// TIA Portal project "Estampado automatizado" (V17)
// Vorlageprojekt für das Buch mit Zielsystem S7-1200

(* hardware
DEVICE "S7-1200-Station_1"  S7-1200 Station
   slot 0: "Baugruppenträger_0"  Rack  V1.0
   slot 1: "PLC_1"  CPU 1211C DC/DC/DC  6ES7 211-1AE40-0XB0  V4.1
*)

// ===== PLC "PLC_1"  CPU 1211C DC/DC/DC =====

VAR_GLOBAL   // PLC tag table "02_Sensores"
   "Sensor_deteccion" AT %I0.3 : Bool;   // Sensor que detecta las bolsas
   "FC X+" AT %I0.4 : Bool;   // Final de carrera del cilindro de impresión extendido
   "FC X-" AT %I0.5 : Bool;   // Final de carrera del cilindro de impresión retraído
   "FC Z+" AT %I0.6 : Bool;   // Final de carrera del cilindro de sellado extendido
   "FC Z-" AT %I0.7 : Bool;   // Final de carrera del cilindro de sellado retraído
   "Sensor_conteo_final" AT %I1.0 : Bool;   // Sensor que detecta las bolsas al final del tunel
END_VAR

VAR_GLOBAL   // PLC tag table "01_Botones y selectores"
   "START" AT %I0.0 : Bool;   // Boton de START
   "STOP" AT %I0.1 : Bool;   // Boton de STOP
   "STOP_EMERGENCIA" AT %I0.2 : Bool;   // Boton enclavado de Parada de Emergencia
   "RESET_CONTEO" AT %I1.1 : Bool;   // Pulsador que reinicia el conteo
END_VAR

VAR_GLOBAL   // PLC tag table "03_Actuadores"
   "Motor_faja" AT %Q0.0 : Bool;   // Motor de la Faja Transportadora
   "EV mov Z" AT %Q0.2 : Bool;   // Electrovalvula Cilindro Eje Z Simple Efecto
   "EV mov X" AT %Q0.1 : Bool;   // Electrovalvula Cilindro Eje X Simple Efecto
   "Motor_faja_2" AT %Q0.6 : Bool;   // Motor de la Faja Transportadora (solo para simulacion)
END_VAR

VAR_GLOBAL   // PLC tag table "04_Luces e indicadores"
   "piloto_start" AT %Q0.3 : Bool;   // Luz indicadora de Proceso en Marcha
   "piloto_stop" AT %Q0.4 : Bool;   // Luz indicadora de Proceso Detenido
   "luz_emergencia" AT %Q0.5 : Bool;   // Luz indicadora de Parada de Emergencia
   "conteo_bolsas" AT %QW30 : Word;   // Cuenta las bolsas que terminan de pasar por el tunel de secado
END_VAR

VAR_GLOBAL   // PLC tag table "00_Variables_de_memoria"
   "Marcha" AT %M0.0 : Bool;   // Variable de memoria Proceso en Marcha
   "E0" AT %M0.1 : Bool;   // Variable de memoria Etapa 0 - inicio
   "E1" AT %M0.2 : Bool;   // Variable de memoria Etapa 1
   "E2" AT %M0.3 : Bool;   // Variable de memoria Etapa 2
   "E3" AT %M0.4 : Bool;   // Variable de memoria Etapa 3
   "E4" AT %M0.5 : Bool;   // Variable de memoria Etapa 4
   "E5" AT %M0.6 : Bool;   // Variable de memoria Etapa 5
   "E6" AT %M0.7 : Bool;   // Variable de memoria Etapa 6
END_VAR

// folder: System blocks/Program resources

DATA_BLOCK "IEC_Counter_0_DB"   // DB1
{ S7_Optimized_Access := 'TRUE' }
AUTHOR : Simatic
FAMILY : IEC
NAME : CNTR
VERSION : 1.0
// stored: InstanceOfName IEC_COUNTER
"IEC_COUNTER"
BEGIN
END_DATA_BLOCK

// folder: (top level)

FUNCTION "MHJ-PLC-Lab-Function-S71200" : Void   // FC9000, SCL
{ S7_Optimized_Access := 'TRUE' }
VERSION : 0.1
   VAR_TEMP
      rdTimeReturn : Int;
      outputTime : DTL;
      SyncVal : Byte;
      forVal : Int;
      forVal_2 : Int;
      Value : Byte;
   END_VAR
   VAR CONSTANT
      CompVal : Byte := 16#34;
      Value_01 : Byte := 16#11;
      Value_01_DW : DWord := 16#A165_D992;
      Value_02_DW : DWord := 16#58BE_4401;
   END_VAR
BEGIN

   #Value:=PEEK(area := 16#82,
        dbNumber := 0,
        byteOffset := 511);
   #Value := #Value + 1;

   POKE(area := 16#82,
        dbNumber := 0,
        byteOffset := 511,
        value := #Value);

   POKE(area:=16#81,
        dbNumber:=0,
        byteOffset:=1016,
        value:=#Value_01_DW);
   POKE(area := 16#81,
        dbNumber := 0,
        byteOffset := 1020,
        value := #Value_02_DW);

   POKE(area := 16#81,
        dbNumber := 0,
        byteOffset := 511,
        value := B#16#00);

   FOR #forVal := 0 TO 120 DO
       FOR #forVal_2:=0 TO 10 DO
           #rdTimeReturn:=RD_SYS_T(#outputTime);
           #rdTimeReturn := WR_SYS_T(#outputTime);
           #rdTimeReturn := RD_SYS_T(#outputTime);
           #rdTimeReturn := WR_SYS_T(#outputTime);
       END_FOR;
       #SyncVal:= PEEK(area := 16#81,
                      dbNumber := 0,
                      byteOffset := 511);
       IF #SyncVal = #CompVal THEN
          GOTO M_1;
       END_IF;
   END_FOR;
   RETURN;

   M_1:
   POKE(area := 16#81,
        dbNumber := 0,
        byteOffset := 511,
        value := B#16#0);
END_FUNCTION

ORGANIZATION_BLOCK "Main"   // OB1, LAD, ProgramCycle
TITLE = "Main Program Sweep (Cycle)"
{ S7_Optimized_Access := 'TRUE' }
VERSION : 0.1
   VAR_INPUT
      Initial_Call : Bool;   // Initial call of this OB
      Remanence : Bool;   // =True, if remanent data are available
   END_VAR
BEGIN

REGION Network 1: Konnektierungsbaustein für PLC-Lab / Bloque de conexion con Factory IO
   // Im Netzwerk 1 wird der Konnektierungsbaustein für PLC-Lab aufgerufen.
   // Dieser Aufruf darf nicht entfernt werden!
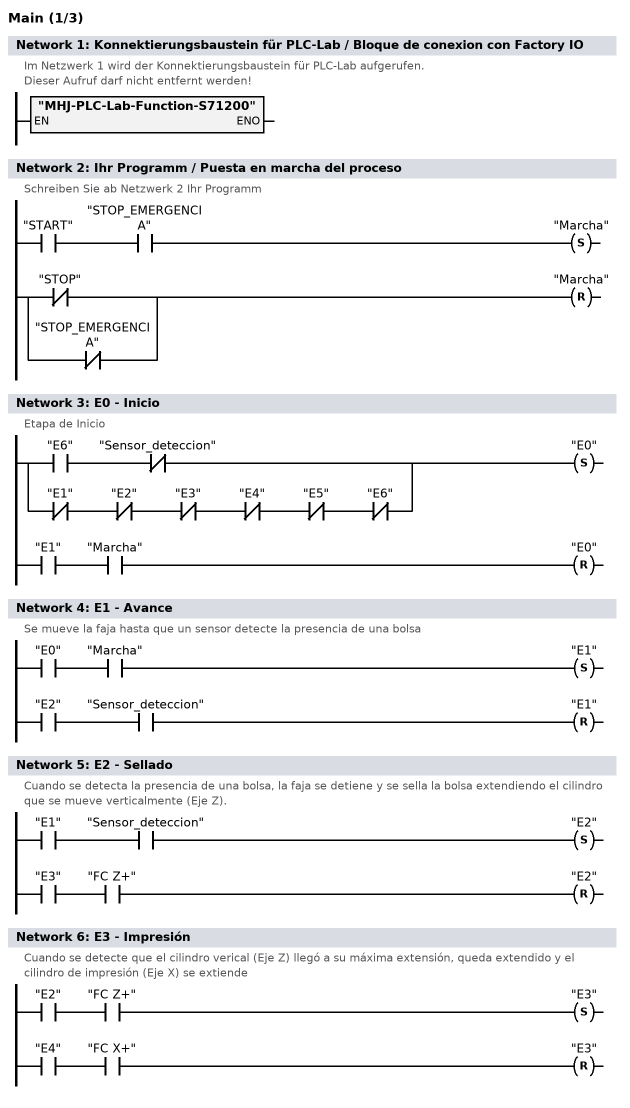
   RUNG wire#powerrail
      "MHJ-PLC-Lab-Function-S71200"()
   END_RUNG
   // the same network as SCL:
   "MHJ-PLC-Lab-Function-S71200"();
END_REGION

REGION Network 2: Ihr Programm / Puesta en marcha del proceso
   // Schreiben Sie ab Netzwerk 2 Ihr Programm
   RUNG wire#powerrail
      Contact( "START" )
      Contact( "STOP_EMERGENCIA" )
      S_Coil( "Marcha" )
   END_RUNG
   RUNG wire#powerrail
      I_Contact( "STOP" )
      wire#w1
      R_Coil( "Marcha" )
   END_RUNG
   RUNG wire#powerrail
      I_Contact( "STOP_EMERGENCIA" )
   END_RUNG wire#w1
   // the same network as SCL:
   IF "START" AND "STOP_EMERGENCIA" THEN "Marcha" := TRUE; END_IF;
   IF NOT "STOP" OR NOT "STOP_EMERGENCIA" THEN "Marcha" := FALSE; END_IF;
END_REGION

REGION Network 3: E0 - Inicio
   // Etapa de Inicio
   RUNG wire#powerrail
      Contact( "E6" )
      I_Contact( "Sensor_deteccion" )
      wire#w1
      S_Coil( "E0" )
   END_RUNG
   RUNG wire#powerrail
      I_Contact( "E1" )
      I_Contact( "E2" )
      I_Contact( "E3" )
      I_Contact( "E4" )
      I_Contact( "E5" )
      I_Contact( "E6" )
   END_RUNG wire#w1
   RUNG wire#powerrail
      Contact( "E1" )
      Contact( "Marcha" )
      R_Coil( "E0" )
   END_RUNG
   // the same network as SCL:
   IF ("E6" AND NOT "Sensor_deteccion") OR (NOT "E1" AND NOT "E2" AND NOT "E3" AND NOT "E4" AND NOT "E5" AND NOT "E6") THEN
       "E0" := TRUE;
   END_IF;
   IF "E1" AND "Marcha" THEN "E0" := FALSE; END_IF;
END_REGION

REGION Network 4: E1 - Avance
   // Se mueve la faja hasta que un sensor detecte la presencia de una bolsa
   RUNG wire#powerrail
      Contact( "E0" )
      Contact( "Marcha" )
      S_Coil( "E1" )
   END_RUNG
   RUNG wire#powerrail
      Contact( "E2" )
      Contact( "Sensor_deteccion" )
      R_Coil( "E1" )
   END_RUNG
   // the same network as SCL:
   IF "E0" AND "Marcha" THEN "E1" := TRUE; END_IF;
   IF "E2" AND "Sensor_deteccion" THEN "E1" := FALSE; END_IF;
END_REGION

REGION Network 5: E2 - Sellado
   // Cuando se detecta la presencia de una bolsa, la faja se detiene y se sella la bolsa extendiendo el cilindro que se mueve verticalmente (Eje Z).
   RUNG wire#powerrail
      Contact( "E1" )
      Contact( "Sensor_deteccion" )
      S_Coil( "E2" )
   END_RUNG
   RUNG wire#powerrail
      Contact( "E3" )
      Contact( "FC Z+" )
      R_Coil( "E2" )
   END_RUNG
   // the same network as SCL:
   IF "E1" AND "Sensor_deteccion" THEN "E2" := TRUE; END_IF;
   IF "E3" AND "FC Z+" THEN "E2" := FALSE; END_IF;
END_REGION

REGION Network 6: E3 - Impresión
   // Cuando se detecte que el cilindro verical (Eje Z) llegó a su máxima extensión, queda extendido y el cilindro de impresión (Eje X) se extiende
   RUNG wire#powerrail
      Contact( "E2" )
      Contact( "FC Z+" )
      S_Coil( "E3" )
   END_RUNG
   RUNG wire#powerrail
      Contact( "E4" )
      Contact( "FC X+" )
      R_Coil( "E3" )
   END_RUNG
   // the same network as SCL:
   IF "E2" AND "FC Z+" THEN "E3" := TRUE; END_IF;
   IF "E4" AND "FC X+" THEN "E3" := FALSE; END_IF;
END_REGION

REGION Network 7: E4 - Retracción Cilindro Impresión Eje X
   // Cuando se detecte que el cilindro de impresión (Eje X) llegó a su máxima extensión, este se vuelve a retraer
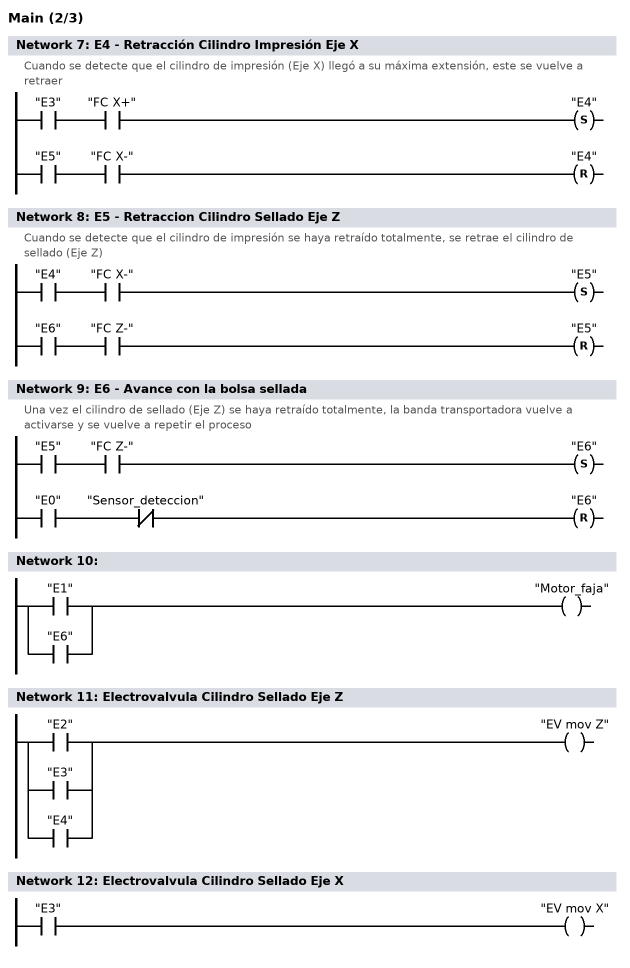
   RUNG wire#powerrail
      Contact( "E3" )
      Contact( "FC X+" )
      S_Coil( "E4" )
   END_RUNG
   RUNG wire#powerrail
      Contact( "E5" )
      Contact( "FC X-" )
      R_Coil( "E4" )
   END_RUNG
   // the same network as SCL:
   IF "E3" AND "FC X+" THEN "E4" := TRUE; END_IF;
   IF "E5" AND "FC X-" THEN "E4" := FALSE; END_IF;
END_REGION

REGION Network 8: E5 - Retraccion Cilindro Sellado Eje Z
   // Cuando se detecte que el cilindro de impresión se haya retraído totalmente, se retrae el cilindro de sellado (Eje Z)
   RUNG wire#powerrail
      Contact( "E4" )
      Contact( "FC X-" )
      S_Coil( "E5" )
   END_RUNG
   RUNG wire#powerrail
      Contact( "E6" )
      Contact( "FC Z-" )
      R_Coil( "E5" )
   END_RUNG
   // the same network as SCL:
   IF "E4" AND "FC X-" THEN "E5" := TRUE; END_IF;
   IF "E6" AND "FC Z-" THEN "E5" := FALSE; END_IF;
END_REGION

REGION Network 9: E6 - Avance con la bolsa sellada
   // Una vez el cilindro de sellado (Eje Z) se haya retraído totalmente, la banda transportadora vuelve a activarse y se vuelve a repetir el proceso
   RUNG wire#powerrail
      Contact( "E5" )
      Contact( "FC Z-" )
      S_Coil( "E6" )
   END_RUNG
   RUNG wire#powerrail
      Contact( "E0" )
      I_Contact( "Sensor_deteccion" )
      R_Coil( "E6" )
   END_RUNG
   // the same network as SCL:
   IF "E5" AND "FC Z-" THEN "E6" := TRUE; END_IF;
   IF "E0" AND NOT "Sensor_deteccion" THEN "E6" := FALSE; END_IF;
END_REGION

REGION Network 10
   RUNG wire#powerrail
      Contact( "E1" )
      wire#w1
      Coil( "Motor_faja" )
   END_RUNG
   RUNG wire#powerrail
      Contact( "E6" )
   END_RUNG wire#w1
   // the same network as SCL:
   "Motor_faja" := "E1" OR "E6";
END_REGION

REGION Network 11: Electrovalvula Cilindro Sellado Eje Z
   RUNG wire#powerrail
      Contact( "E2" )
      wire#w1
      Coil( "EV mov Z" )
   END_RUNG
   RUNG wire#powerrail
      Contact( "E3" )
   END_RUNG wire#w1
   RUNG wire#powerrail
      Contact( "E4" )
   END_RUNG wire#w1
   // the same network as SCL:
   "EV mov Z" := "E2" OR "E3" OR "E4";
END_REGION

REGION Network 12: Electrovalvula Cilindro Sellado Eje X
   RUNG wire#powerrail
      Contact( "E3" )
      Coil( "EV mov X" )
   END_RUNG
   // the same network as SCL:
   "EV mov X" := "E3";
END_REGION

REGION Network 13: Pilotos e indicadores
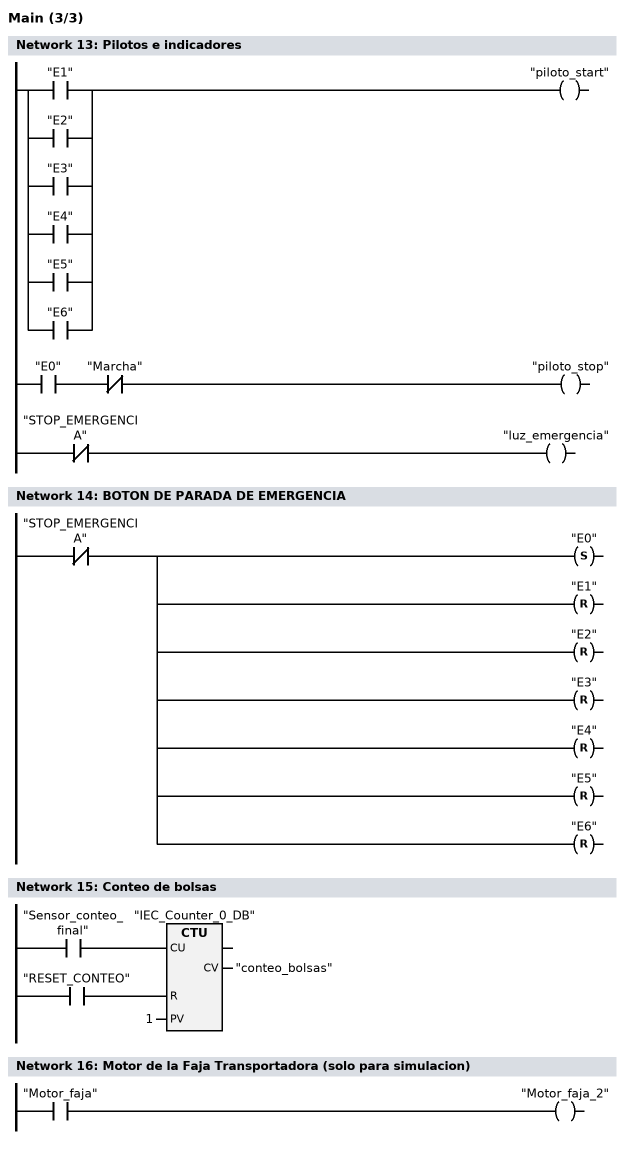
   RUNG wire#powerrail
      Contact( "E1" )
      wire#w1
      Coil( "piloto_start" )
   END_RUNG
   RUNG wire#powerrail
      Contact( "E2" )
   END_RUNG wire#w1
   RUNG wire#powerrail
      Contact( "E3" )
   END_RUNG wire#w1
   RUNG wire#powerrail
      Contact( "E4" )
   END_RUNG wire#w1
   RUNG wire#powerrail
      Contact( "E5" )
   END_RUNG wire#w1
   RUNG wire#powerrail
      Contact( "E6" )
   END_RUNG wire#w1
   RUNG wire#powerrail
      Contact( "E0" )
      I_Contact( "Marcha" )
      Coil( "piloto_stop" )
   END_RUNG
   RUNG wire#powerrail
      I_Contact( "STOP_EMERGENCIA" )
      Coil( "luz_emergencia" )
   END_RUNG
   // the same network as SCL:
   "piloto_start" := "E1" OR "E2" OR "E3" OR "E4" OR "E5" OR "E6";
   "piloto_stop" := "E0" AND NOT "Marcha";
   "luz_emergencia" := NOT "STOP_EMERGENCIA";
END_REGION

REGION Network 14: BOTON DE PARADA DE EMERGENCIA
   RUNG wire#powerrail
      I_Contact( "STOP_EMERGENCIA" )
      wire#w1
      S_Coil( "E0" )
   END_RUNG
   RUNG wire#w1
      R_Coil( "E1" )
   END_RUNG
   RUNG wire#w1
      R_Coil( "E2" )
   END_RUNG
   RUNG wire#w1
      R_Coil( "E3" )
   END_RUNG
   RUNG wire#w1
      R_Coil( "E4" )
   END_RUNG
   RUNG wire#w1
      R_Coil( "E5" )
   END_RUNG
   RUNG wire#w1
      R_Coil( "E6" )
   END_RUNG
   // the same network as SCL:
   IF NOT "STOP_EMERGENCIA" THEN
       "E0" := TRUE;
       "E1" := FALSE;
       "E2" := FALSE;
       "E3" := FALSE;
       "E4" := FALSE;
       "E5" := FALSE;
       "E6" := FALSE;
   END_IF;
END_REGION

REGION Network 15: Conteo de bolsas
   "IEC_Counter_0_DB".CTU(CU := "Sensor_conteo_final", R := "RESET_CONTEO", PV := 1, CV => "conteo_bolsas");
END_REGION

REGION Network 16: Motor de la Faja Transportadora (solo para simulacion)
   RUNG wire#powerrail
      Contact( "Motor_faja" )
      Coil( "Motor_faja_2" )
   END_RUNG
   // the same network as SCL:
   "Motor_faja_2" := "Motor_faja";
END_REGION
END_ORGANIZATION_BLOCK